FUNCTION_BLOCK fb_BusPingEvent
VAR_INPUT
	 I_sID         			:STRING(10);     // Geräte-ID (z.B. '12345')
	 I_sReceivedString		:STRING(255);	
	 I_bReset				:BOOL;
END_VAR
VAR_OUTPUT
	Q_bOut					:BOOL;
END_VAR
VAR
	findString0				:STRING ;
	findString1				:STRING ;
	findString2				:STRING ;
	findString3				:STRING ;
	findString4				:STRING ;
	findString5				:STRING ;	// Für CYD Ping
END_VAR

(* Wenn ein Taster gedrückt wird *)
findString0 := CONCAT(I_sID,'.');
findString0 := CONCAT(findString0,'BTN');
findString0 := CONCAT(findString0,'.');

(* Wenn ein Relais geschaltet wird *)
findString1 := CONCAT(I_sID,'.');
findString1 := CONCAT(findString1,'OUT');
findString1 := CONCAT(findString1,'.');

(* Wenn Ein Temperatur Event Kommt *)
findString2 := CONCAT(I_sID,'.');
findString2 := CONCAT(findString2,'TMP.1.');

(* Wenn Ein Feuchtigkeit Event Kommt *)
findString3 := CONCAT(I_sID,'.');
findString3 := CONCAT(findString3,'RHD.1.');

(* Wenn Ein Helligkeit Event Kommt *)
findString4 := CONCAT(I_sID,'.');
findString4 := CONCAT(findString4,'BRS.1.');

(* Wenn Ein Display Helligkeits Event Kommt für CYD *)
findString5 := CONCAT(I_sID,'.');
findString5 := CONCAT(findString5,'LBN.16.');

IF I_bReset
THEN
	Q_bOut := FALSE;
ELSE
	IF 	FIND(I_sReceivedString,findString0) >0 
		OR FIND(I_sReceivedString,findString1) >0 
		OR FIND(I_sReceivedString,findString2) >0 
		OR FIND(I_sReceivedString,findString3) >0 
		OR FIND(I_sReceivedString,findString4) >0 
		OR FIND(I_sReceivedString,findString5) >0 
	THEN
		Q_bOut := TRUE;
	ELSE
		Q_bOut := FALSE;
	END_IF
END_IF

END_FUNCTION_BLOCK

(* stored: Version 1.1.0.1, ProductVersion 3.1.4024.12
   POU fb_BusPingEvent: Id {b07ed474-f0db-45c9-bf2c-2641b67dcd51}, SpecialFunc None *)
